# EPICS alarm handler configuration: caQtDM_UnitTests/tst_qtcontrols/fixtures/alh/include_loop.alhConfig
GROUP NULL LOOP
INCLUDE LOOP include_loop.alhConfig
CHANNEL LOOP loop:ch
